# EPICS substitutions: evrSupport/Db/ioc/evrPatternXL16.substitutions
#
# Pattern records
file evrPatternAll.db {
#	    Device        ,  SLC Pattern Check LNK    , EVR/Trigger
#	                                                  Links
  pattern { DEVICE        ,        LINK4              , LINK5 , LINK6 , TREF }
	  { IOC:XL16:EV01 ,         ""                ,  ""   ,  ""   , 1E06 }
}
# Event records
file evrEventAll.db {
  pattern { DEVICE   , TREF }
	  { IOC:XL16:EV01, 1E06 }
}
